// TIA Portal project "create_dataset_tia_portal" (V17)

(* hardware
DEVICE "S7-1500/ET200MP station_1"  S7-1500 station
   slot 0: "Rail_0"  Rack  6ES7 590-1***0-0AA0
   slot 1: "PLC_1"  CPU 1513-1 PN  6ES7 513-1AL01-0AB0  V2.6
      slot 3: "CPU display_1"  6ES7591-1AA00-0AA0
      slot 32768: "PROFINET interface_1"  X1
         slot 32769: "Port_1"  X1 P1
         slot 32770: "Port_2"  X1 P2
*)

// ===== PLC "PLC_1"  CPU 1513-1 PN =====

VAR_GLOBAL   // PLC tag table "Default tag table"
   "OPC_START" AT %I0.0 : Bool;
   "OPC_STOP" AT %I0.1 : Bool;
   "SISTEM" AT %M0.0 : Bool;
   "OPC_EMITTER" AT %Q0.0 : Bool;
   "OPC_BELT_LONG" AT %QD2 : Real;
   "OPC_CAPACITIVE_1" AT %I0.2 : Bool;
   "OPC_CAM" AT %QD6 : DInt;
   "OPC_PHOTOELECTRICO" AT %I0.3 : Bool;
   "UNITS_TRIG" AT %M0.1 : Bool;
   "2_UNITS" AT %M0.2 : Bool;
   "OPC_GATE_1" AT %Q0.1 : Bool;
   "OPC_GATE_2" AT %Q0.2 : Bool;
   "OPC_PISTON_SENSOR" AT %I0.4 : Bool;
   "OPC_BELT_FINALE" AT %Q0.3 : Bool;
   "OPC_PISTON" AT %QD10 : Real;
   "OPC_CAPACITIVE_2" AT %I0.5 : Bool;
   "ACTIVATE_BELT_FINALE" AT %M0.5 : Bool;
   "OPC_GATE_FINALE" AT %Q0.4 : Bool;
   "OPC_CAPACITIVE_3" AT %I0.6 : Bool;
   "OPC_PISTON_SAMPLES" AT %Q0.6 : Bool;
   "OPC_PISTON_SAMPLES_SENSOR" AT %I1.2 : Bool;
END_VAR

DATA_BLOCK "IEC_Timer_0_DB"   // DB1
{ S7_Optimized_Access := 'TRUE' }
AUTHOR : Simatic
FAMILY : IEC
NAME : IEC_TMR
VERSION : 1.0
// stored: InstanceOfName IEC_TIMER
"IEC_TIMER"
BEGIN
END_DATA_BLOCK

DATA_BLOCK "IEC_Counter_0_DB"   // DB2
{ S7_Optimized_Access := 'TRUE' }
AUTHOR : Simatic
FAMILY : IEC
NAME : CNTR
VERSION : 1.0
// stored: InstanceOfName IEC_COUNTER
"IEC_COUNTER"
BEGIN
END_DATA_BLOCK

DATA_BLOCK "CONFIG_VARS"   // DB7
{ S7_Optimized_Access := 'TRUE' }
VERSION : 0.1
   VAR
      EMITTER_CONFIG : Bool;
      "COUNTER" : Int;
      TRIG_4_PY_INSTRUCTION : Bool;
      INSTRUCTION_2_PY : Bool;
      PY_RESPONSE : Bool;
      CONFIG_END : Bool;
      TRIG_N : Bool;
      INSTRUCTION_TRIG_N : Bool;
      GATE_FINALE : Bool;
      N_TRIG_FOR_EMITTER : Bool;
   END_VAR
BEGIN
END_DATA_BLOCK

// folder: System blocks/Program resources

DATA_BLOCK "IEC_Timer_0_DB_3"   // DB3
{ S7_Optimized_Access := 'TRUE' }
AUTHOR : Simatic
FAMILY : IEC
NAME : IEC_TMR
VERSION : 1.0
// stored: InstanceOfName IEC_TIMER
"IEC_TIMER"
BEGIN
END_DATA_BLOCK

// folder: (top level)

FUNCTION "SAMPLE" : Void   // FC2, LAD
{ S7_Optimized_Access := 'TRUE' }
VERSION : 0.1
   VAR_TEMP
      EMITTER_CONFIG : Bool;
      EMITTER_CONFIG_1 : Bool;
      EMITTER_CONFIG_2 : Bool;
   END_VAR
   VAR_TEMP   // added for the SCL form of the ladder/FBD networks
      _w1 : Bool;
      _w2 : Bool;
      _w3 : Bool;
   END_VAR
BEGIN

REGION Network 1
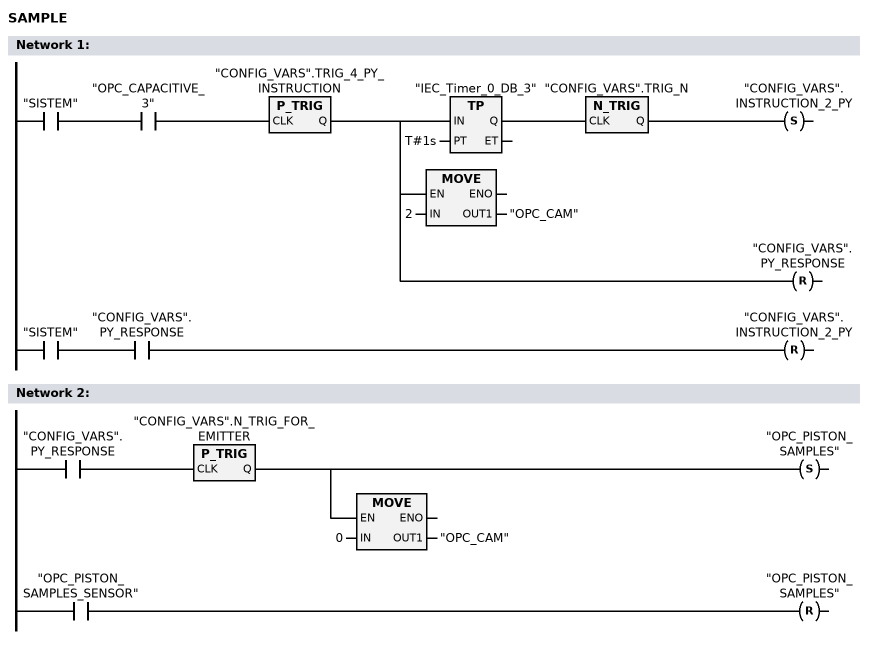
   #_w1 := "SISTEM" AND "OPC_CAPACITIVE_3";
   #_w2 := #_w1 AND NOT "CONFIG_VARS".TRIG_4_PY_INSTRUCTION;   // rising edge
   "CONFIG_VARS".TRIG_4_PY_INSTRUCTION := #_w1;
   "IEC_Timer_0_DB_3".TP(IN := #_w2, PT := T#1s);
   #_w3 := NOT "IEC_Timer_0_DB_3".Q AND "CONFIG_VARS".TRIG_N;   // falling edge
   "CONFIG_VARS".TRIG_N := "IEC_Timer_0_DB_3".Q;
   IF #_w3 THEN "CONFIG_VARS".INSTRUCTION_2_PY := TRUE; END_IF;
   IF #_w2 THEN
       "OPC_CAM" := 2;
       "CONFIG_VARS".PY_RESPONSE := FALSE;
   END_IF;
   IF "SISTEM" AND "CONFIG_VARS".PY_RESPONSE THEN "CONFIG_VARS".INSTRUCTION_2_PY := FALSE; END_IF;
END_REGION

REGION Network 2
   RUNG wire#powerrail
      Contact( "CONFIG_VARS".PY_RESPONSE )
      P_Trig( "CONFIG_VARS".N_TRIG_FOR_EMITTER )
      wire#w1
      S_Coil( "OPC_PISTON_SAMPLES" )
   END_RUNG
   RUNG wire#w1
      Move(in := 0, out1 => "OPC_CAM")
   END_RUNG
   RUNG wire#powerrail
      Contact( "OPC_PISTON_SAMPLES_SENSOR" )
      R_Coil( "OPC_PISTON_SAMPLES" )
   END_RUNG
   // the same network as SCL:
   #_w1 := "CONFIG_VARS".PY_RESPONSE AND NOT "CONFIG_VARS".N_TRIG_FOR_EMITTER;   // rising edge
   "CONFIG_VARS".N_TRIG_FOR_EMITTER := "CONFIG_VARS".PY_RESPONSE;
   IF #_w1 THEN
       "OPC_PISTON_SAMPLES" := TRUE;
       "OPC_CAM" := 0;
   END_IF;
   IF "OPC_PISTON_SAMPLES_SENSOR" THEN "OPC_PISTON_SAMPLES" := FALSE; END_IF;
END_REGION
END_FUNCTION

ORGANIZATION_BLOCK "Main"   // OB1, LAD, ProgramCycle
TITLE = "Main Program Sweep (Cycle)"
{ S7_Optimized_Access := 'TRUE' }
VERSION : 0.1
   VAR_INPUT
      Initial_Call : Bool;   // Initial call of this OB
      Remanence : Bool;   // =True, if remanent data are available
   END_VAR
   VAR_TEMP   // added for the SCL form of the ladder/FBD networks
      _w1 : Bool;
      _w2 : Bool;
   END_VAR
BEGIN

REGION Network 1: Arranque y parada del proceso
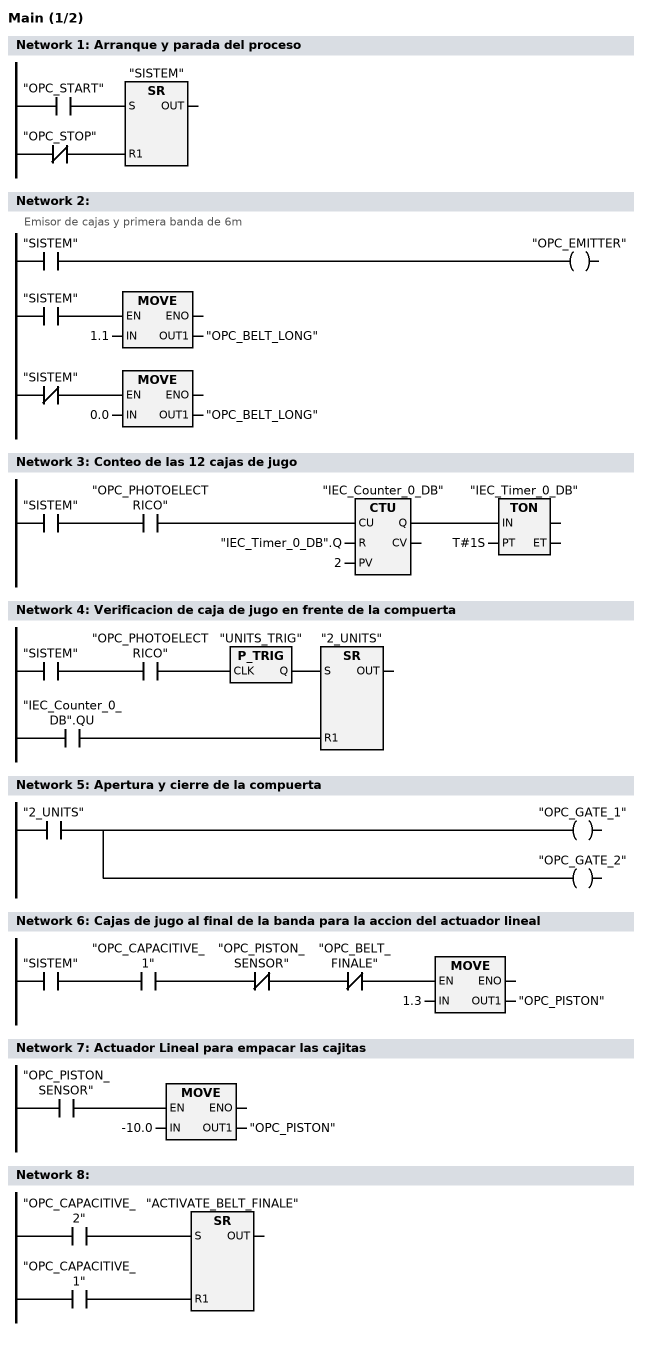
   RUNG wire#powerrail
      Contact( "OPC_START" )
      S_SR(operand := "SISTEM", r1 := wire#w1)
   END_RUNG
   RUNG wire#powerrail
      I_Contact( "OPC_STOP" )
   END_RUNG wire#w1
   // the same network as SCL:
   IF "OPC_START" THEN
       "SISTEM" := TRUE;   // SR flip-flop
   END_IF;
   IF NOT "OPC_STOP" THEN "SISTEM" := FALSE; END_IF;
END_REGION

REGION Network 2
   // Emisor de cajas y primera banda de 6m
   RUNG wire#powerrail
      Contact( "SISTEM" )
      Coil( "OPC_EMITTER" )
   END_RUNG
   RUNG wire#powerrail
      Contact( "SISTEM" )
      Move(in := 1.1, out1 => "OPC_BELT_LONG")
   END_RUNG
   RUNG wire#powerrail
      I_Contact( "SISTEM" )
      Move(in := 0.0, out1 => "OPC_BELT_LONG")
   END_RUNG
   // the same network as SCL:
   "OPC_EMITTER" := "SISTEM";
   IF "SISTEM" THEN "OPC_BELT_LONG" := 1.1; END_IF;
   IF NOT "SISTEM" THEN "OPC_BELT_LONG" := 0.0; END_IF;
END_REGION

REGION Network 3: Conteo de las 12 cajas de jugo
   "IEC_Counter_0_DB".CTU(CU := "SISTEM" AND "OPC_PHOTOELECTRICO", R := "IEC_Timer_0_DB".Q, PV := 2);
   "IEC_Timer_0_DB".TON(IN := "IEC_Counter_0_DB".Q, PT := T#1S);
END_REGION

REGION Network 4: Verificacion de caja de jugo en frente de la compuerta
   RUNG wire#powerrail
      Contact( "SISTEM" )
      Contact( "OPC_PHOTOELECTRICO" )
      P_Trig( "UNITS_TRIG" )
      S_SR(operand := "2_UNITS", r1 := wire#w1)
   END_RUNG
   RUNG wire#powerrail
      Contact( "IEC_Counter_0_DB".QU )
   END_RUNG wire#w1
   // the same network as SCL:
   #_w1 := "SISTEM" AND "OPC_PHOTOELECTRICO";
   #_w2 := #_w1 AND NOT "UNITS_TRIG";   // rising edge
   "UNITS_TRIG" := #_w1;
   IF #_w2 THEN
       "2_UNITS" := TRUE;   // SR flip-flop
   END_IF;
   IF "IEC_Counter_0_DB".QU THEN "2_UNITS" := FALSE; END_IF;
END_REGION

REGION Network 5: Apertura y cierre de la compuerta
   RUNG wire#powerrail
      Contact( "2_UNITS" )
      wire#w1
      Coil( "OPC_GATE_1" )
   END_RUNG
   RUNG wire#w1
      Coil( "OPC_GATE_2" )
   END_RUNG
   // the same network as SCL:
   "OPC_GATE_1" := "2_UNITS";
   "OPC_GATE_2" := "2_UNITS";
END_REGION

REGION Network 6: Cajas de jugo al final de la banda para la accion del actuador lineal
   RUNG wire#powerrail
      Contact( "SISTEM" )
      Contact( "OPC_CAPACITIVE_1" )
      I_Contact( "OPC_PISTON_SENSOR" )
      I_Contact( "OPC_BELT_FINALE" )
      Move(in := 1.3, out1 => "OPC_PISTON")
   END_RUNG
   // the same network as SCL:
   IF "SISTEM" AND "OPC_CAPACITIVE_1" AND NOT "OPC_PISTON_SENSOR" AND NOT "OPC_BELT_FINALE" THEN
       "OPC_PISTON" := 1.3;
   END_IF;
END_REGION

REGION Network 7: Actuador Lineal para empacar las cajitas
   RUNG wire#powerrail
      Contact( "OPC_PISTON_SENSOR" )
      Move(in := -10.0, out1 => "OPC_PISTON")
   END_RUNG
   // the same network as SCL:
   IF "OPC_PISTON_SENSOR" THEN "OPC_PISTON" := -10.0; END_IF;
END_REGION

REGION Network 8
   RUNG wire#powerrail
      Contact( "OPC_CAPACITIVE_2" )
      S_SR(operand := "ACTIVATE_BELT_FINALE", r1 := wire#w1)
   END_RUNG
   RUNG wire#powerrail
      Contact( "OPC_CAPACITIVE_1" )
   END_RUNG wire#w1
   // the same network as SCL:
   IF "OPC_CAPACITIVE_2" THEN
       "ACTIVATE_BELT_FINALE" := TRUE;   // SR flip-flop
   END_IF;
   IF "OPC_CAPACITIVE_1" THEN "ACTIVATE_BELT_FINALE" := FALSE; END_IF;
END_REGION

REGION Network 9: Detencion y Movimiento de la segunda banda en base a la posicion de la Caja grande
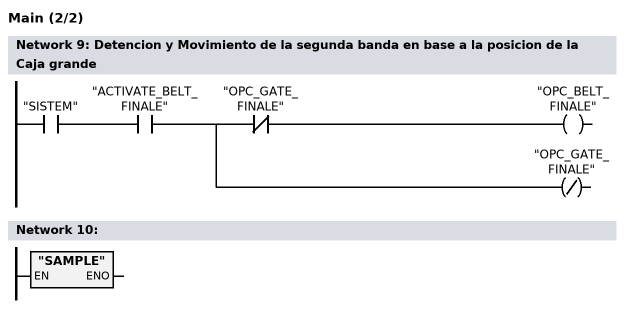
   RUNG wire#powerrail
      Contact( "SISTEM" )
      Contact( "ACTIVATE_BELT_FINALE" )
      wire#w1
      I_Contact( "OPC_GATE_FINALE" )
      Coil( "OPC_BELT_FINALE" )
   END_RUNG
   RUNG wire#w1
      I_Coil( "OPC_GATE_FINALE" )
   END_RUNG
   // the same network as SCL:
   #_w1 := "SISTEM" AND "ACTIVATE_BELT_FINALE";
   "OPC_BELT_FINALE" := #_w1 AND NOT "OPC_GATE_FINALE";
   "OPC_GATE_FINALE" := NOT #_w1;
END_REGION

REGION Network 10
   RUNG wire#powerrail
      "SAMPLE"()
   END_RUNG
   // the same network as SCL:
   "SAMPLE"();
END_REGION
END_ORGANIZATION_BLOCK